(* IEC 61131-3 sources: horner-cscape-mcp/artifacts/exports, 4 files *)

(* ---- test_unit_project.st ---- *)
(* ============================================================================ *)
(* Consolidated Structured Text POU Bundle: test_unit_project *)
(* Export Format: IEC 61131-3 Pure Structured Text *)
(* Exported At: 2026-09-06T22:29:34.523620+00:00 *)
(* Hardware Lockout: Enforced (Simulation Only) *)
(* ============================================================================ *)

(* ---------------------------------------------------------------------------- *)
(* POU: FB_ConveyorTest (FB_ConveyorTest.st) *)
(* ---------------------------------------------------------------------------- *)
FUNCTION_BLOCK FB_ConveyorTest
VAR_INPUT
    RunCmd : BOOL;
    PE_Sensor : BOOL;
END_VAR
VAR_OUTPUT
    MotorOut : BOOL;
    BoxCount : INT := 0;
END_VAR
IF RunCmd THEN
    MotorOut := TRUE;
    IF PE_Sensor THEN
        BoxCount := BoxCount + 1;
    END_IF;
ELSE
    MotorOut := FALSE;
END_IF;
END_FUNCTION_BLOCK

(* ---- test_unit_project_consolidated.st ---- *)
(* ========================================== *)
(* Project: test_unit_project                      *)
(* Target PLC: T5RTI *)
(* Exported at: 2026-09-04T05:52:29.070619+00:00                     *)
(* ========================================== *)

(* --- POU: FB_ConveyorTest --- *)
FUNCTION_BLOCK FB_ConveyorTest
VAR_INPUT
    RunCmd : BOOL;
    PE_Sensor : BOOL;
END_VAR
VAR_OUTPUT
    MotorOut : BOOL;
    BoxCount : INT := 0;
END_VAR
IF RunCmd THEN
    MotorOut := TRUE;
    IF PE_Sensor THEN
        BoxCount := BoxCount + 1;
    END_IF;
ELSE
    MotorOut := FALSE;
END_IF;
END_FUNCTION_BLOCK

(* ---- E2E_ClosedLoop_Verification.st ---- *)
(* ============================================================================ *)
(* Consolidated Structured Text POU Bundle: E2E_ClosedLoop_Verification *)
(* Export Format: IEC 61131-3 Pure Structured Text *)
(* Exported At: 2026-09-06T22:29:33.746050+00:00 *)
(* Hardware Lockout: Enforced (Simulation Only) *)
(* ============================================================================ *)

(* ---------------------------------------------------------------------------- *)
(* POU: ClosedLoopTank (ClosedLoopTank.st) *)
(* ---------------------------------------------------------------------------- *)
PROGRAM ClosedLoopTank
VAR_INPUT
    RawLevelIn : INT;
    SetPoint : REAL := 50.0;
    AutoMode : BOOL := TRUE;
END_VAR
VAR_OUTPUT
    PumpSpeed : INT;
    HighAlarm : BOOL;
END_VAR
VAR
    LevelPercent : REAL;
END_VAR

LevelPercent := (INT_TO_REAL(RawLevelIn) / 32000.0) * 100.0;

IF LevelPercent >= 90.0 THEN
    HighAlarm := TRUE;
ELSE
    HighAlarm := FALSE;
END_IF;

IF AutoMode THEN
    IF LevelPercent < SetPoint THEN
        PumpSpeed := 25000;
    ELSE
        PumpSpeed := 8000;
    END_IF;
ELSE
    PumpSpeed := 0;
END_IF;
END_PROGRAM

(* ---- ExportMCPProofProj.st ---- *)
(* ============================================================================ *)
(* Consolidated Structured Text POU Bundle: ExportMCPProofProj *)
(* Export Format: IEC 61131-3 Pure Structured Text *)
(* Exported At: 2026-09-09T03:39:07.645970+00:00 *)
(* Hardware Lockout: Enforced (Simulation Only) *)
(* ============================================================================ *)

(* ---------------------------------------------------------------------------- *)
(* POU: ProofPOU (ProofPOU.st) *)
(* ---------------------------------------------------------------------------- *)
PROGRAM ProofPOU
VAR
    nCount : INT := 0;
    bFlag : BOOL := TRUE;
END_VAR
nCount := nCount + 1;
END_PROGRAM
